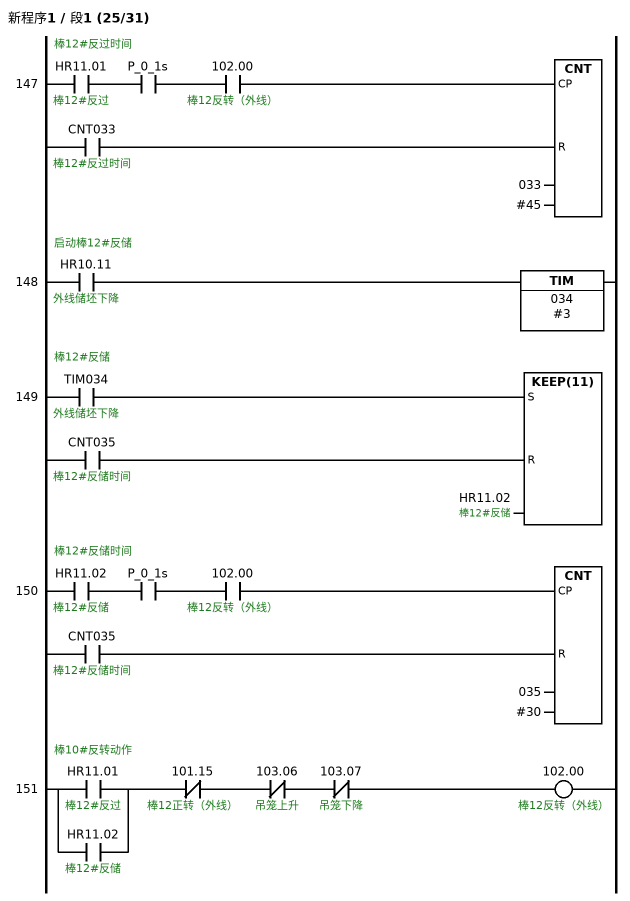
; [picture p24: 新程序1 / 段1, rungs 147-151]
; rung 147: 棒12#反过时间
LD HR11.01  ; 棒12#反过
AND P_0_1s
AND 102.00  ; 棒12反转（外线）
LD CNT033  ; 棒12#反过时间
CNT 033 #45
; rung 148: 启动棒12#反储
LD HR10.11  ; 外线储坯下降
TIM 034 #3
; rung 149: 棒12#反储
LD TIM034  ; 外线储坯下降
LD CNT035  ; 棒12#反储时间
KEEP(11) HR11.02  ; 棒12#反储
; rung 150: 棒12#反储时间
LD HR11.02  ; 棒12#反储
AND P_0_1s
AND 102.00  ; 棒12反转（外线）
LD CNT035  ; 棒12#反储时间
CNT 035 #30
; rung 151: 棒10#反转动作
LD HR11.01  ; 棒12#反过
OR HR11.02  ; 棒12#反储
ANDNOT 101.15  ; 棒12正转（外线）
ANDNOT 103.06  ; 吊笼上升
ANDNOT 103.07  ; 吊笼下降
OUT 102.00  ; 棒12反转（外线）

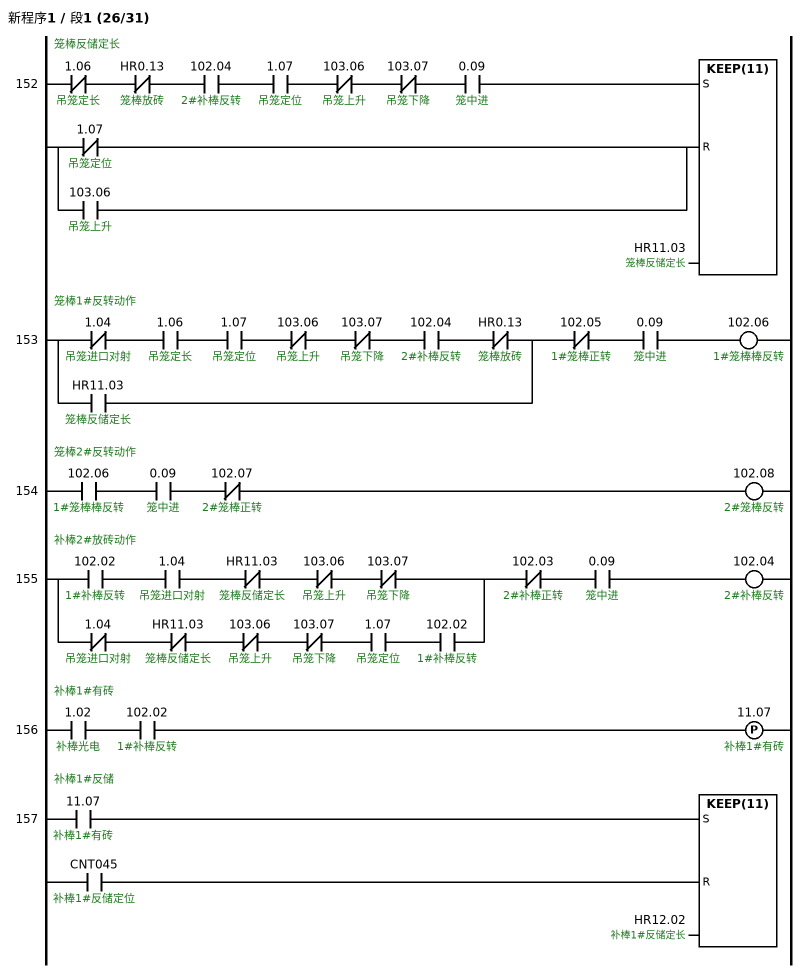
; rung 152: 笼棒反储定长
LDNOT 1.06  ; 吊笼定长
ANDNOT HR0.13  ; 笼棒放砖
AND 102.04  ; 2#补棒反转
AND 1.07  ; 吊笼定位
ANDNOT 103.06  ; 吊笼上升
ANDNOT 103.07  ; 吊笼下降
AND 0.09  ; 笼中进
LDNOT 1.07  ; 吊笼定位
OR 103.06  ; 吊笼上升
KEEP(11) HR11.03  ; 笼棒反储定长
; rung 153: 笼棒1#反转动作
LDNOT 1.04  ; 吊笼进口对射
AND 1.06  ; 吊笼定长
AND 1.07  ; 吊笼定位
ANDNOT 103.06  ; 吊笼上升
ANDNOT 103.07  ; 吊笼下降
AND 102.04  ; 2#补棒反转
ANDNOT HR0.13  ; 笼棒放砖
OR HR11.03  ; 笼棒反储定长
ANDNOT 102.05  ; 1#笼棒正转
AND 0.09  ; 笼中进
OUT 102.06  ; 1#笼棒棒反转
; rung 154: 笼棒2#反转动作
LD 102.06  ; 1#笼棒棒反转
AND 0.09  ; 笼中进
ANDNOT 102.07  ; 2#笼棒正转
OUT 102.08  ; 2#笼棒反转
; rung 155: 补棒2#放砖动作
LD 102.02  ; 1#补棒反转
AND 1.04  ; 吊笼进口对射
ANDNOT HR11.03  ; 笼棒反储定长
ANDNOT 103.06  ; 吊笼上升
ANDNOT 103.07  ; 吊笼下降
LDNOT 1.04  ; 吊笼进口对射
ANDNOT HR11.03  ; 笼棒反储定长
ANDNOT 103.06  ; 吊笼上升
ANDNOT 103.07  ; 吊笼下降
AND 1.07  ; 吊笼定位
AND 102.02  ; 1#补棒反转
ORLD
ANDNOT 102.03  ; 2#补棒正转
AND 0.09  ; 笼中进
OUT 102.04  ; 2#补棒反转
; rung 156: 补棒1#有砖
LD 1.02  ; 补棒光电
AND 102.02  ; 1#补棒反转
DIFU(13) 11.07  ; 补棒1#有砖
; rung 157: 补棒1#反储
LD 11.07  ; 补棒1#有砖
LD CNT045  ; 补棒1#反储定位
KEEP(11) HR12.02  ; 补棒1#反储定长

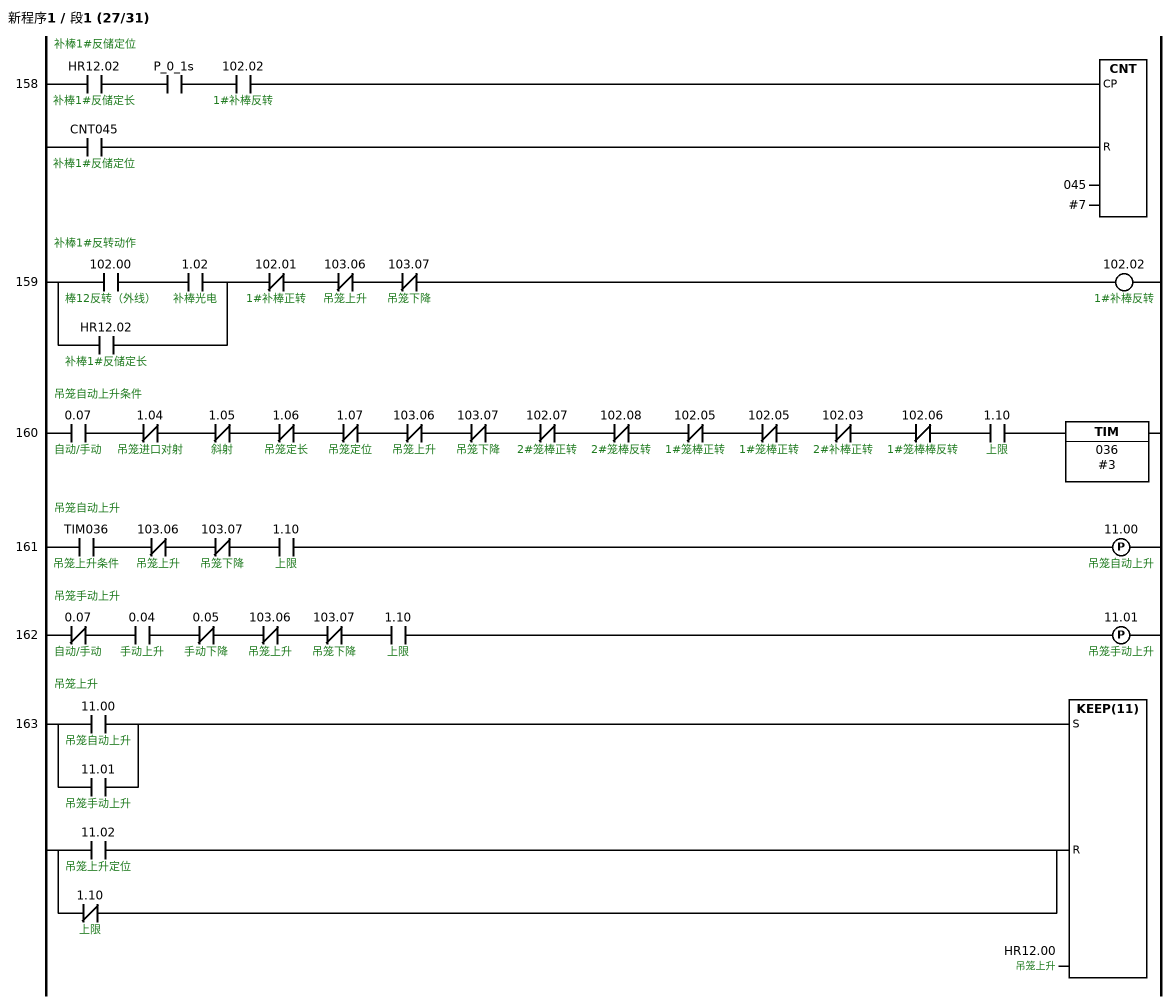
; rung 158: 补棒1#反储定位
LD HR12.02  ; 补棒1#反储定长
AND P_0_1s
AND 102.02  ; 1#补棒反转
LD CNT045  ; 补棒1#反储定位
CNT 045 #7
; rung 159: 补棒1#反转动作
LD 102.00  ; 棒12反转（外线）
AND 1.02  ; 补棒光电
OR HR12.02  ; 补棒1#反储定长
ANDNOT 102.01  ; 1#补棒正转
ANDNOT 103.06  ; 吊笼上升
ANDNOT 103.07  ; 吊笼下降
OUT 102.02  ; 1#补棒反转
; rung 160: 吊笼自动上升条件
LD 0.07  ; 自动/手动
ANDNOT 1.04  ; 吊笼进口对射
ANDNOT 1.05  ; 斜射
ANDNOT 1.06  ; 吊笼定长
ANDNOT 1.07  ; 吊笼定位
ANDNOT 103.06  ; 吊笼上升
ANDNOT 103.07  ; 吊笼下降
ANDNOT 102.07  ; 2#笼棒正转
ANDNOT 102.08  ; 2#笼棒反转
ANDNOT 102.05  ; 1#笼棒正转
ANDNOT 102.05  ; 1#笼棒正转
ANDNOT 102.03  ; 2#补棒正转
ANDNOT 102.06  ; 1#笼棒棒反转
AND 1.10  ; 上限
TIM 036 #3
; rung 161: 吊笼自动上升
LD TIM036  ; 吊笼上升条件
ANDNOT 103.06  ; 吊笼上升
ANDNOT 103.07  ; 吊笼下降
AND 1.10  ; 上限
DIFU(13) 11.00  ; 吊笼自动上升
; rung 162: 吊笼手动上升
LDNOT 0.07  ; 自动/手动
AND 0.04  ; 手动上升
ANDNOT 0.05  ; 手动下降
ANDNOT 103.06  ; 吊笼上升
ANDNOT 103.07  ; 吊笼下降
AND 1.10  ; 上限
DIFU(13) 11.01  ; 吊笼手动上升
; rung 163: 吊笼上升
LD 11.00  ; 吊笼自动上升
OR 11.01  ; 吊笼手动上升
LD 11.02  ; 吊笼上升定位
ORNOT 1.10  ; 上限
KEEP(11) HR12.00  ; 吊笼上升

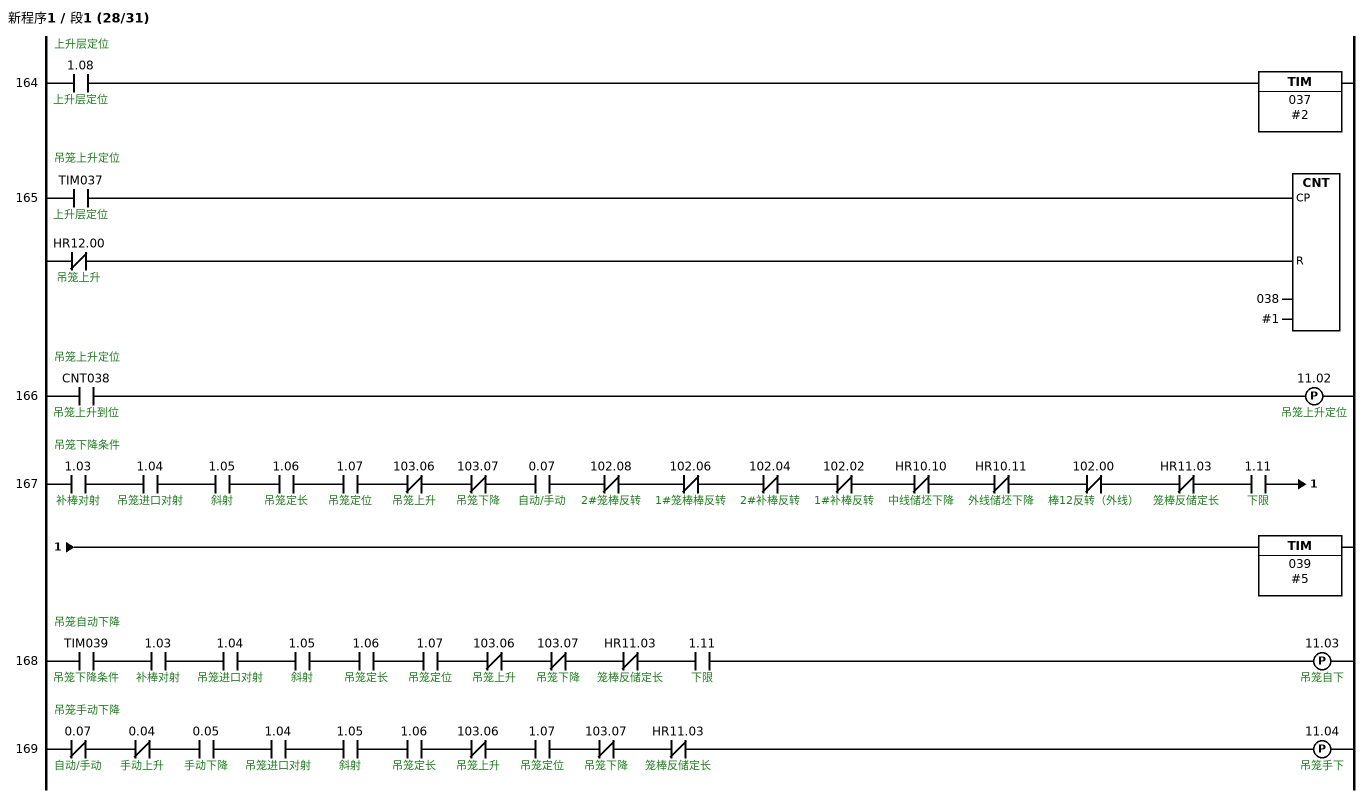
; rung 164: 上升层定位
LD 1.08  ; 上升层定位
TIM 037 #2
; rung 165: 吊笼上升定位
LD TIM037  ; 上升层定位
LDNOT HR12.00  ; 吊笼上升
CNT 038 #1
; rung 166: 吊笼上升定位
LD CNT038  ; 吊笼上升到位
DIFU(13) 11.02  ; 吊笼上升定位
; rung 167: 吊笼下降条件
LD 1.03  ; 补棒对射
AND 1.04  ; 吊笼进口对射
AND 1.05  ; 斜射
AND 1.06  ; 吊笼定长
AND 1.07  ; 吊笼定位
ANDNOT 103.06  ; 吊笼上升
ANDNOT 103.07  ; 吊笼下降
AND 0.07  ; 自动/手动
ANDNOT 102.08  ; 2#笼棒反转
ANDNOT 102.06  ; 1#笼棒棒反转
ANDNOT 102.04  ; 2#补棒反转
ANDNOT 102.02  ; 1#补棒反转
ANDNOT HR10.10  ; 中线储坯下降
ANDNOT HR10.11  ; 外线储坯下降
ANDNOT 102.00  ; 棒12反转（外线）
ANDNOT HR11.03  ; 笼棒反储定长
AND 1.11  ; 下限
TIM 039 #5
; rung 168: 吊笼自动下降
LD TIM039  ; 吊笼下降条件
AND 1.03  ; 补棒对射
AND 1.04  ; 吊笼进口对射
AND 1.05  ; 斜射
AND 1.06  ; 吊笼定长
AND 1.07  ; 吊笼定位
ANDNOT 103.06  ; 吊笼上升
ANDNOT 103.07  ; 吊笼下降
ANDNOT HR11.03  ; 笼棒反储定长
AND 1.11  ; 下限
DIFU(13) 11.03  ; 吊笼自下
; rung 169: 吊笼手动下降
LDNOT 0.07  ; 自动/手动
ANDNOT 0.04  ; 手动上升
AND 0.05  ; 手动下降
AND 1.04  ; 吊笼进口对射
AND 1.05  ; 斜射
AND 1.06  ; 吊笼定长
ANDNOT 103.06  ; 吊笼上升
AND 1.07  ; 吊笼定位
ANDNOT 103.07  ; 吊笼下降
ANDNOT HR11.03  ; 笼棒反储定长
DIFU(13) 11.04  ; 吊笼手下

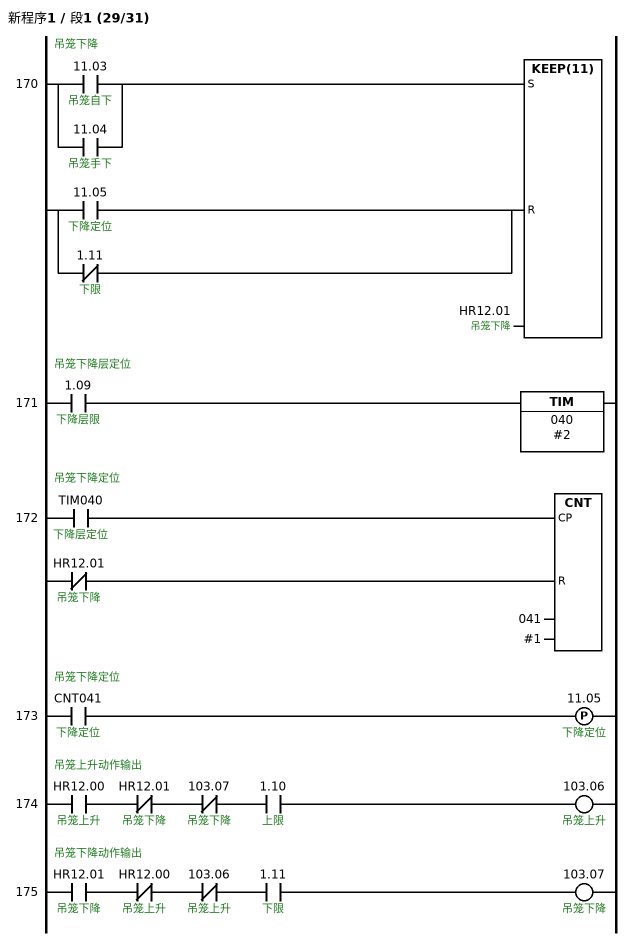
; rung 170: 吊笼下降
LD 11.03  ; 吊笼自下
OR 11.04  ; 吊笼手下
LD 11.05  ; 下降定位
ORNOT 1.11  ; 下限
KEEP(11) HR12.01  ; 吊笼下降
; rung 171: 吊笼下降层定位
LD 1.09  ; 下降层限
TIM 040 #2
; rung 172: 吊笼下降定位
LD TIM040  ; 下降层定位
LDNOT HR12.01  ; 吊笼下降
CNT 041 #1
; rung 173: 吊笼下降定位
LD CNT041  ; 下降定位
DIFU(13) 11.05  ; 下降定位
; rung 174: 吊笼上升动作输出
LD HR12.00  ; 吊笼上升
ANDNOT HR12.01  ; 吊笼下降
ANDNOT 103.07  ; 吊笼下降
AND 1.10  ; 上限
OUT 103.06  ; 吊笼上升
; rung 175: 吊笼下降动作输出
LD HR12.01  ; 吊笼下降
ANDNOT HR12.00  ; 吊笼上升
ANDNOT 103.06  ; 吊笼上升
AND 1.11  ; 下限
OUT 103.07  ; 吊笼下降

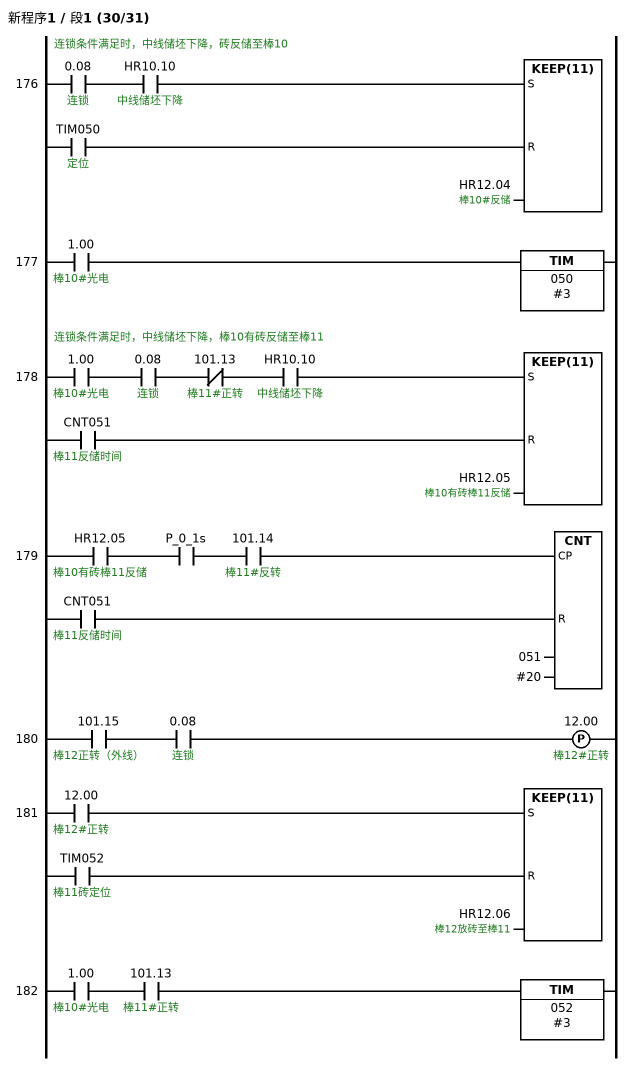
; rung 176: 连锁条件满足时，中线储坯下降，砖反储至棒10
LD 0.08  ; 连锁
AND HR10.10  ; 中线储坯下降
LD TIM050  ; 定位
KEEP(11) HR12.04  ; 棒10#反储
; rung 177
LD 1.00  ; 棒10#光电
TIM 050 #3
; rung 178: 连锁条件满足时，中线储坯下降，棒10有砖反储至棒11
LD 1.00  ; 棒10#光电
AND 0.08  ; 连锁
ANDNOT 101.13  ; 棒11#正转
AND HR10.10  ; 中线储坯下降
LD CNT051  ; 棒11反储时间
KEEP(11) HR12.05  ; 棒10有砖棒11反储
; rung 179
LD HR12.05  ; 棒10有砖棒11反储
AND P_0_1s
AND 101.14  ; 棒11#反转
LD CNT051  ; 棒11反储时间
CNT 051 #20
; rung 180
LD 101.15  ; 棒12正转（外线）
AND 0.08  ; 连锁
DIFU(13) 12.00  ; 棒12#正转
; rung 181
LD 12.00  ; 棒12#正转
LD TIM052  ; 棒11砖定位
KEEP(11) HR12.06  ; 棒12放砖至棒11
; rung 182
LD 1.00  ; 棒10#光电
AND 101.13  ; 棒11#正转
TIM 052 #3

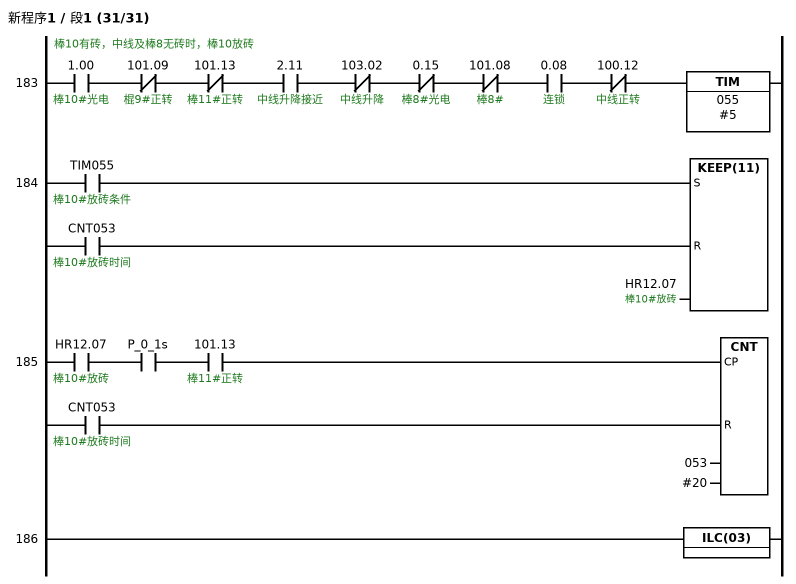
; rung 183: 棒10有砖，中线及棒8无砖时，棒10放砖
LD 1.00  ; 棒10#光电
ANDNOT 101.09  ; 棍9#正转
ANDNOT 101.13  ; 棒11#正转
AND 2.11  ; 中线升降接近
ANDNOT 103.02  ; 中线升降
ANDNOT 0.15  ; 棒8#光电
ANDNOT 101.08  ; 棒8#
AND 0.08  ; 连锁
ANDNOT 100.12  ; 中线正转
TIM 055 #5
; rung 184
LD TIM055  ; 棒10#放砖条件
LD CNT053  ; 棒10#放砖时间
KEEP(11) HR12.07  ; 棒10#放砖
; rung 185
LD HR12.07  ; 棒10#放砖
AND P_0_1s
AND 101.13  ; 棒11#正转
LD CNT053  ; 棒10#放砖时间
CNT 053 #20
; rung 186
ILC(03)
; rung 187
END(01)